RoboDK station: 6640_station.rdk

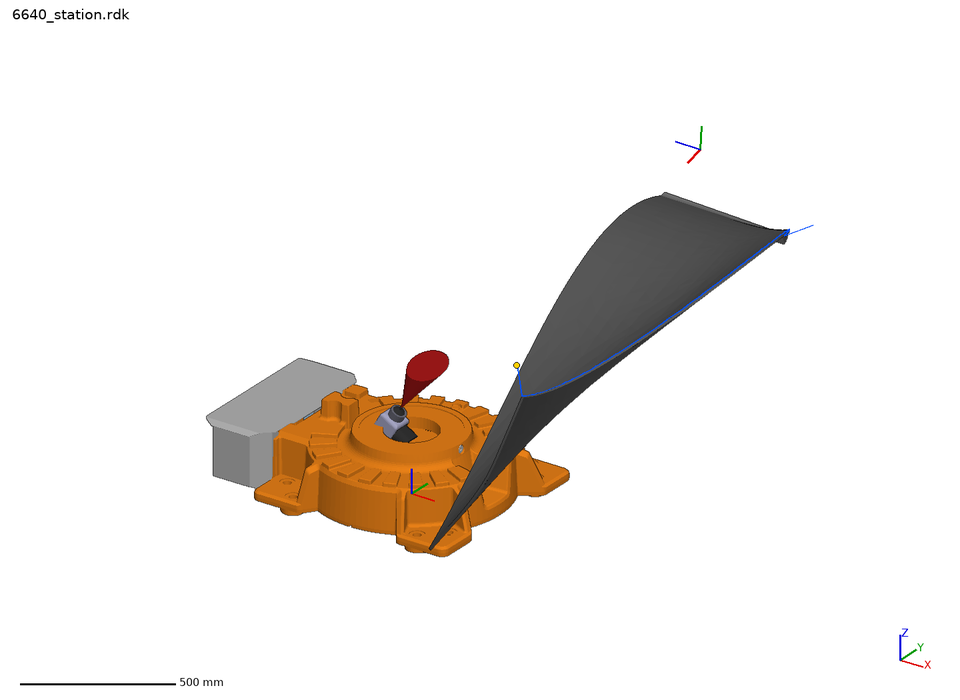
[picture v0: the station drawn from its stored meshes, robots at their saved joint values, targets as dots, program paths as lines]
Station 6640_station (saved by RoboDK 5.3.2). Poses are relative to the parent item; angles as X-Y-Z fixed-axis rotations.
  - frame Frame 2 at (435.15, 997.23, 955.19) mm, rotated rx 84.12 ry 5.86 rz -82.67 deg
    - object Curve_sparse at (0, 0, 0) mm
    - object generic_fan_blade at (0, 0, 0) mm, size 1633.1 x 757.5 x 617.2 mm, 1 curves, geometry from generic_fan_blade.igs
  - machining project Path1 settings: rotZ(0) | rotX(0)*rotY(0) | rotz(0)
  - program Path1 (113 instructions, listed below)
  - frame ABB IRB 6640-180/2.55 Base at (0, 0, 0) mm
    - robot ABB IRB 6640-180/2.55: 6 axes, payload 180 kg, reach 2550 mm, repeatability 0.07 mm, weight 1310 kg
        joint limits [-170, -65, -180, -300, -120, -360] to [170, 85, 70, 300, 120, 360]; home [0, 0, 0, 0, 0, 0]; saved at [53.767, 31.077, 10.307, -34.616, 114.864, 62.566]
      - tool Paint gun, TCP at (75, 0, 493.3) mm, rotated rx 0 ry 30 rz 0 deg, size 203.2 x 279.7 x 471.5 mm
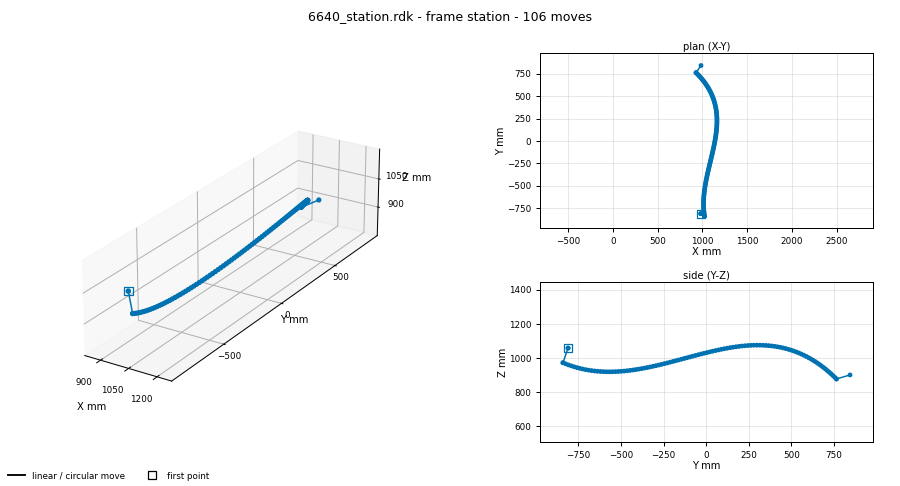
[picture p0: tool path of 6640_station.rdk in frame station, 106 of 106 moves have a stored position in this frame; points joined in program order, loops and branches not executed]

--- program Path1 (robot ABB IRB 6640-180/2.55) ---
  Smooth(1)
  Set speed (500.0 mm/s)
  Set Ref.: Frame 2
  Set Tool: Paint gun
  Show Paint gun
  MoveJ 1 to (1843, 323.42, -278.71) mm, rotated rx -160.29 ry -61.06 rz -82.99 deg; joints [-55.097, -38.535, 54.626, 57.641, 41.418, -99.137]
  MoveL 2 to (1843, 323.42, -278.71) mm, rotated rx -160.29 ry -61.06 rz -82.99 deg; joints [-55.097, -38.535, 54.626, 57.641, 41.418, -99.137]
  MoveL 3 to (1886.54, 245.77, -324.26) mm, rotated rx -160.29 ry -61.06 rz -82.99 deg; joints [-53.957, -33.784, 56.818, 64.848, 37.125, -107.941]
  MoveL 4 to (1886.54, 245.77, -324.26) mm, rotated rx -160.29 ry -61.06 rz -82.99 deg; joints [-53.957, -33.784, 56.818, 64.848, 37.125, -107.941]
  Set speed (50.0 mm/s)
  MoveL 5 to (1871.02, 237.56, -324.78) mm, rotated rx -160.62 ry -60.74 rz -83.73 deg; joints [-53.875, -34.314, 57.338, 64.8, 37.71, -106.973]
  MoveL 6 to (1855.29, 229.78, -325.6) mm, rotated rx -160.63 ry -60.92 rz -84.77 deg; joints [-53.458, -34.858, 57.629, 63.666, 37.945, -104.885]
  MoveL 7 to (1839.38, 222.45, -326.7) mm, rotated rx -160.51 ry -61.31 rz -85.95 deg; joints [-52.891, -35.379, 57.794, 62.071, 38.083, -102.301]
  MoveL 8 to (1823.28, 215.57, -328.1) mm, rotated rx -160.35 ry -61.75 rz -87.2 deg; joints [-52.27, -35.863, 57.894, 60.357, 38.247, -99.564]
  MoveL 9 to (1807.02, 209.15, -329.78) mm, rotated rx -160.22 ry -62.19 rz -88.46 deg; joints [-51.64, -36.309, 57.963, 58.692, 38.477, -96.847]
  MoveL 10 to (1790.62, 203.19, -331.75) mm, rotated rx -160.11 ry -62.58 rz -89.71 deg; joints [-51.014, -36.722, 58.014, 57.137, 38.778, -94.214]
  MoveL 11 to (1774.08, 197.71, -334) mm, rotated rx -160.03 ry -62.95 rz -90.94 deg; joints [-50.391, -37.105, 58.048, 55.697, 39.138, -91.674]
  MoveL 12 to (1757.44, 192.71, -336.52) mm, rotated rx -159.97 ry -63.29 rz -92.16 deg; joints [-49.767, -37.458, 58.065, 54.358, 39.543, -89.215]
  MoveL 13 to (1740.71, 188.17, -339.31) mm, rotated rx -159.93 ry -63.62 rz -93.37 deg; joints [-49.135, -37.783, 58.062, 53.107, 39.982, -86.827]
  MoveL 14 to (1723.9, 184.11, -342.35) mm, rotated rx -159.91 ry -63.94 rz -94.57 deg; joints [-48.493, -38.081, 58.041, 51.935, 40.446, -84.505]
  MoveL 15 to (1707.03, 180.51, -345.64) mm, rotated rx -159.9 ry -64.25 rz -95.74 deg; joints [-47.841, -38.354, 58.002, 50.844, 40.929, -82.253]
  MoveL 16 to (1690.11, 177.36, -349.16) mm, rotated rx -159.91 ry -64.54 rz -96.89 deg; joints [-47.181, -38.607, 57.951, 49.84, 41.423, -80.08]
  MoveL 17 to (1673.17, 174.65, -352.91) mm, rotated rx -159.93 ry -64.82 rz -98 deg; joints [-46.514, -38.843, 57.892, 48.927, 41.92, -77.993]
  MoveL 18 to (1656.22, 172.37, -356.87) mm, rotated rx -159.97 ry -65.08 rz -99.08 deg; joints [-45.841, -39.067, 57.83, 48.104, 42.414, -75.993]
  MoveL 19 to (1639.26, 170.51, -361.03) mm, rotated rx -160.03 ry -65.31 rz -100.1 deg; joints [-45.161, -39.285, 57.767, 47.369, 42.896, -74.079]
  MoveL 20 to (1622.3, 169.06, -365.37) mm, rotated rx -160.12 ry -65.52 rz -101.08 deg; joints [-44.472, -39.497, 57.703, 46.71, 43.36, -72.243]
  MoveL 21 to (1605.37, 167.99, -369.89) mm, rotated rx -160.21 ry -65.72 rz -102.02 deg; joints [-43.772, -39.707, 57.639, 46.115, 43.802, -70.472]
  MoveL 22 to (1588.46, 167.28, -374.56) mm, rotated rx -160.31 ry -65.9 rz -102.91 deg; joints [-43.056, -39.912, 57.571, 45.567, 44.218, -68.753]
  MoveL 23 to (1571.57, 166.93, -379.39) mm, rotated rx -160.42 ry -66.08 rz -103.76 deg; joints [-42.322, -40.111, 57.497, 45.052, 44.607, -67.07]
  MoveL 24 to (1554.73, 166.92, -384.35) mm, rotated rx -160.52 ry -66.26 rz -104.59 deg; joints [-41.567, -40.302, 57.413, 44.554, 44.969, -65.412]
  MoveL 25 to (1537.92, 167.22, -389.43) mm, rotated rx -160.62 ry -66.44 rz -105.39 deg; joints [-40.788, -40.481, 57.315, 44.061, 45.306, -63.767]
  MoveL 26 to (1521.16, 167.82, -394.63) mm, rotated rx -160.7 ry -66.64 rz -106.16 deg; joints [-39.985, -40.646, 57.2, 43.565, 45.618, -62.128]
  MoveL 27 to (1504.44, 168.7, -399.93) mm, rotated rx -160.77 ry -66.85 rz -106.93 deg; joints [-39.156, -40.793, 57.067, 43.059, 45.908, -60.489]
  MoveL 28 to (1487.77, 169.85, -405.32) mm, rotated rx -160.81 ry -67.07 rz -107.68 deg; joints [-38.303, -40.92, 56.914, 42.54, 46.178, -58.848]
  MoveL 29 to (1471.14, 171.25, -410.79) mm, rotated rx -160.84 ry -67.31 rz -108.42 deg; joints [-37.425, -41.027, 56.741, 42.003, 46.429, -57.204]
  MoveL 30 to (1454.56, 172.87, -416.33) mm, rotated rx -160.85 ry -67.57 rz -109.15 deg; joints [-36.523, -41.112, 56.547, 41.45, 46.662, -55.556]
  MoveL 31 to (1438.02, 174.71, -421.93) mm, rotated rx -160.84 ry -67.85 rz -109.87 deg; joints [-35.599, -41.175, 56.332, 40.879, 46.88, -53.905]
  MoveL 32 to (1421.52, 176.76, -427.59) mm, rotated rx -160.8 ry -68.15 rz -110.58 deg; joints [-34.653, -41.215, 56.098, 40.289, 47.083, -52.251]
  MoveL 33 to (1405.07, 178.98, -433.29) mm, rotated rx -160.74 ry -68.46 rz -111.29 deg; joints [-33.687, -41.233, 55.843, 39.681, 47.273, -50.595]
  MoveL 34 to (1388.64, 181.38, -439.03) mm, rotated rx -160.65 ry -68.79 rz -111.99 deg; joints [-32.7, -41.226, 55.57, 39.054, 47.452, -48.938]
  MoveL 35 to (1372.25, 183.93, -444.79) mm, rotated rx -160.53 ry -69.13 rz -112.69 deg; joints [-31.695, -41.197, 55.277, 38.407, 47.62, -47.278]
  MoveL 36 to (1355.89, 186.62, -450.58) mm, rotated rx -160.38 ry -69.49 rz -113.38 deg; joints [-30.672, -41.144, 54.965, 37.74, 47.779, -45.618]
  MoveL 37 to (1339.56, 189.43, -456.38) mm, rotated rx -160.21 ry -69.87 rz -114.08 deg; joints [-29.632, -41.067, 54.635, 37.053, 47.93, -43.956]
  MoveL 38 to (1323.25, 192.36, -462.18) mm, rotated rx -160 ry -70.26 rz -114.78 deg; joints [-28.575, -40.967, 54.287, 36.345, 48.075, -42.293]
  MoveL 39 to (1306.95, 195.39, -467.98) mm, rotated rx -159.75 ry -70.66 rz -115.49 deg; joints [-27.502, -40.844, 53.922, 35.616, 48.215, -40.629]
  MoveL 40 to (1290.67, 198.51, -473.78) mm, rotated rx -159.46 ry -71.08 rz -116.19 deg; joints [-26.414, -40.7, 53.54, 34.866, 48.349, -38.964]
  MoveL 41 to (1274.4, 201.7, -479.55) mm, rotated rx -159.13 ry -71.51 rz -116.91 deg; joints [-25.311, -40.534, 53.143, 34.094, 48.48, -37.298]
  MoveL 42 to (1258.13, 204.96, -485.31) mm, rotated rx -158.76 ry -71.95 rz -117.64 deg; joints [-24.193, -40.348, 52.731, 33.299, 48.607, -35.631]
  MoveL 43 to (1241.86, 208.26, -491.03) mm, rotated rx -158.34 ry -72.4 rz -118.38 deg; joints [-23.06, -40.142, 52.305, 32.48, 48.731, -33.961]
  MoveL 44 to (1225.59, 211.59, -496.72) mm, rotated rx -157.87 ry -72.86 rz -119.13 deg; joints [-21.913, -39.918, 51.865, 31.635, 48.854, -32.288]
  MoveL 45 to (1209.31, 214.96, -502.37) mm, rotated rx -157.34 ry -73.33 rz -119.91 deg; joints [-20.751, -39.674, 51.411, 30.762, 48.976, -30.609]
  MoveL 46 to (1193.01, 218.33, -507.96) mm, rotated rx -156.74 ry -73.81 rz -120.72 deg; joints [-19.573, -39.41, 50.943, 29.859, 49.101, -28.923]
  MoveL 47 to (1176.7, 221.7, -513.5) mm, rotated rx -156.06 ry -74.3 rz -121.57 deg; joints [-18.38, -39.125, 50.46, 28.924, 49.23, -27.228]
  MoveL 48 to (1160.36, 225.06, -518.97) mm, rotated rx -155.3 ry -74.8 rz -122.47 deg; joints [-17.171, -38.817, 49.96, 27.954, 49.368, -25.521]
  MoveL 49 to (1143.99, 228.39, -524.37) mm, rotated rx -154.43 ry -75.31 rz -123.43 deg; joints [-15.945, -38.485, 49.444, 26.947, 49.517, -23.803]
  MoveL 50 to (1127.58, 231.68, -529.68) mm, rotated rx -153.43 ry -75.84 rz -124.48 deg; joints [-14.703, -38.128, 48.909, 25.901, 49.682, -22.07]
  MoveL 51 to (1111.14, 234.91, -534.91) mm, rotated rx -152.29 ry -76.39 rz -125.63 deg; joints [-13.443, -37.744, 48.356, 24.815, 49.865, -20.322]
  MoveL 52 to (1094.65, 238.08, -540.05) mm, rotated rx -150.98 ry -76.94 rz -126.9 deg; joints [-12.166, -37.332, 47.783, 23.688, 50.069, -18.558]
  MoveL 53 to (1078.12, 241.17, -545.07) mm, rotated rx -149.48 ry -77.51 rz -128.33 deg; joints [-10.869, -36.894, 47.192, 22.517, 50.296, -16.776]
  MoveL 54 to (1061.53, 244.16, -549.99) mm, rotated rx -147.74 ry -78.08 rz -129.93 deg; joints [-9.554, -36.43, 46.584, 21.302, 50.548, -14.977]
  MoveL 55 to (1044.89, 247.05, -554.77) mm, rotated rx -145.74 ry -78.65 rz -131.75 deg; joints [-8.217, -35.94, 45.959, 20.042, 50.825, -13.157]
  MoveL 56 to (1028.18, 249.8, -559.43) mm, rotated rx -143.44 ry -79.22 rz -133.81 deg; joints [-6.858, -35.426, 45.32, 18.734, 51.128, -11.317]
  MoveL 57 to (1011.42, 252.41, -563.94) mm, rotated rx -140.79 ry -79.78 rz -136.17 deg; joints [-5.475, -34.889, 44.668, 17.377, 51.457, -9.454]
  MoveL 58 to (994.59, 254.86, -568.29) mm, rotated rx -137.74 ry -80.32 rz -138.86 deg; joints [-4.066, -34.331, 44.004, 15.968, 51.814, -7.566]
  MoveL 59 to (977.7, 257.14, -572.47) mm, rotated rx -134.25 ry -80.84 rz -141.93 deg; joints [-2.631, -33.752, 43.33, 14.505, 52.2, -5.65]
  MoveL 60 to (960.73, 259.22, -576.48) mm, rotated rx -130.25 ry -81.31 rz -145.43 deg; joints [-1.166, -33.15, 42.647, 12.986, 52.617, -3.707]
  MoveL 61 to (943.7, 261.09, -580.29) mm, rotated rx -125.71 ry -81.74 rz -149.4 deg; joints [0.328, -32.525, 41.955, 11.411, 53.071, -1.733]
  MoveL 62 to (926.6, 262.73, -583.9) mm, rotated rx -120.59 ry -82.12 rz -153.88 deg; joints [1.854, -31.875, 41.255, 9.778, 53.564, 0.271]
  MoveL 63 to (909.44, 264.11, -587.29) mm, rotated rx -114.89 ry -82.42 rz -158.86 deg; joints [3.412, -31.196, 40.547, 8.088, 54.104, 2.305]
  MoveL 64 to (892.21, 265.22, -590.45) mm, rotated rx -108.65 ry -82.63 rz -164.3 deg; joints [5.002, -30.488, 39.831, 6.342, 54.694, 4.368]
  MoveL 65 to (874.92, 266.04, -593.36) mm, rotated rx -102 ry -82.75 rz -170.06 deg; joints [6.624, -29.747, 39.109, 4.543, 55.339, 6.458]
  MoveL 66 to (857.57, 266.55, -596) mm, rotated rx -95.12 ry -82.76 rz -175.97 deg; joints [8.279, -28.973, 38.381, 2.694, 56.043, 8.572]
  MoveL 67 to (840.18, 266.73, -598.37) mm, rotated rx -88.24 ry -82.65 rz 178.22 deg; joints [9.965, -28.163, 37.652, 0.799, 56.808, 10.708]
  MoveL 68 to (822.75, 266.54, -600.45) mm, rotated rx -81.6 ry -82.44 rz 172.75 deg; joints [11.681, -27.319, 36.924, -1.137, 57.637, 12.86]
  MoveL 69 to (805.3, 265.99, -602.22) mm, rotated rx -75.41 ry -82.12 rz 167.81 deg; joints [13.425, -26.439, 36.201, -3.106, 58.53, 15.025]
  MoveL 70 to (787.84, 265.04, -603.67) mm, rotated rx -69.79 ry -81.71 rz 163.55 deg; joints [15.194, -25.523, 35.487, -5.102, 59.486, 17.197]
  MoveL 71 to (770.37, 263.68, -604.78) mm, rotated rx -64.79 ry -81.22 rz 160 deg; joints [16.983, -24.572, 34.786, -7.116, 60.505, 19.368]
  MoveL 72 to (752.93, 261.89, -605.55) mm, rotated rx -60.41 ry -80.68 rz 157.15 deg; joints [18.788, -23.585, 34.102, -9.137, 61.587, 21.53]
  MoveL 73 to (735.53, 259.66, -605.96) mm, rotated rx -56.59 ry -80.09 rz 154.96 deg; joints [20.601, -22.561, 33.436, -11.153, 62.731, 23.675]
  MoveL 74 to (718.19, 256.98, -606) mm, rotated rx -53.27 ry -79.47 rz 153.35 deg; joints [22.417, -21.497, 32.792, -13.152, 63.935, 25.792]
  MoveL 75 to (700.94, 253.83, -605.66) mm, rotated rx -50.36 ry -78.83 rz 152.23 deg; joints [24.226, -20.393, 32.169, -15.119, 65.198, 27.871]
  MoveL 76 to (683.78, 250.21, -604.94) mm, rotated rx -47.79 ry -78.17 rz 151.53 deg; joints [26.021, -19.246, 31.568, -17.041, 66.517, 29.903]
  MoveL 77 to (666.76, 246.11, -603.84) mm, rotated rx -45.51 ry -77.49 rz 151.18 deg; joints [27.792, -18.054, 30.988, -18.904, 67.89, 31.878]
  MoveL 78 to (649.88, 241.54, -602.35) mm, rotated rx -43.44 ry -76.8 rz 151.11 deg; joints [29.532, -16.817, 30.429, -20.696, 69.313, 33.788]
  MoveL 79 to (633.17, 236.5, -600.48) mm, rotated rx -41.55 ry -76.09 rz 151.26 deg; joints [31.231, -15.531, 29.887, -22.404, 70.783, 35.626]
  MoveL 80 to (616.66, 230.99, -598.23) mm, rotated rx -39.79 ry -75.37 rz 151.59 deg; joints [32.883, -14.196, 29.36, -24.02, 72.297, 37.386]
  MoveL 81 to (600.36, 225.03, -595.61) mm, rotated rx -38.12 ry -74.63 rz 152.04 deg; joints [34.48, -12.809, 28.842, -25.533, 73.852, 39.065]
  MoveL 82 to (584.29, 218.62, -592.63) mm, rotated rx -36.52 ry -73.86 rz 152.6 deg; joints [36.016, -11.366, 28.328, -26.936, 75.447, 40.66]
  MoveL 83 to (568.46, 211.78, -589.29) mm, rotated rx -34.96 ry -73.05 rz 153.23 deg; joints [37.486, -9.867, 27.815, -28.224, 77.081, 42.172]
  MoveL 84 to (552.91, 204.52, -585.61) mm, rotated rx -33.43 ry -72.21 rz 153.93 deg; joints [38.885, -8.31, 27.296, -29.395, 78.751, 43.601]
  MoveL 85 to (537.62, 196.87, -581.6) mm, rotated rx -31.92 ry -71.31 rz 154.67 deg; joints [40.212, -6.698, 26.771, -30.446, 80.453, 44.952]
  MoveL 86 to (522.62, 188.84, -577.28) mm, rotated rx -30.45 ry -70.38 rz 155.47 deg; joints [41.464, -5.035, 26.24, -31.381, 82.18, 46.231]
  MoveL 87 to (507.91, 180.46, -572.66) mm, rotated rx -29.03 ry -69.4 rz 156.33 deg; joints [42.642, -3.329, 25.704, -32.204, 83.922, 47.445]
  MoveL 88 to (493.49, 171.73, -567.76) mm, rotated rx -27.66 ry -68.39 rz 157.26 deg; joints [43.748, -1.59, 25.168, -32.921, 85.669, 48.603]
  MoveL 89 to (479.36, 162.69, -562.59) mm, rotated rx -26.35 ry -67.35 rz 158.25 deg; joints [44.785, 0.174, 24.636, -33.539, 87.412, 49.712]
  MoveL 90 to (465.53, 153.35, -557.16) mm, rotated rx -25.11 ry -66.3 rz 159.3 deg; joints [45.754, 1.957, 24.108, -34.063, 89.146, 50.779]
  MoveL 91 to (451.98, 143.72, -551.51) mm, rotated rx -23.91 ry -65.21 rz 160.41 deg; joints [46.658, 3.76, 23.581, -34.499, 90.874, 51.811]
  MoveL 92 to (438.73, 133.83, -545.62) mm, rotated rx -22.76 ry -64.09 rz 161.56 deg; joints [47.498, 5.584, 23.054, -34.847, 92.6, 52.813]
  MoveL 93 to (425.75, 123.7, -539.53) mm, rotated rx -21.64 ry -62.94 rz 162.77 deg; joints [48.275, 7.433, 22.521, -35.112, 94.329, 53.793]
  MoveL 94 to (413.06, 113.33, -533.24) mm, rotated rx -20.56 ry -61.74 rz 164.03 deg; joints [48.991, 9.304, 21.984, -35.296, 96.062, 54.756]
  MoveL 95 to (400.64, 102.75, -526.77) mm, rotated rx -19.52 ry -60.52 rz 165.34 deg; joints [49.648, 11.188, 21.447, -35.405, 97.793, 55.711]
  MoveL 96 to (388.49, 91.97, -520.13) mm, rotated rx -18.52 ry -59.28 rz 166.7 deg; joints [50.253, 13.076, 20.916, -35.446, 99.511, 56.663]
  MoveL 97 to (376.59, 81, -513.32) mm, rotated rx -17.57 ry -58.02 rz 168.12 deg; joints [50.808, 14.961, 20.395, -35.424, 101.212, 57.617]
  MoveL 98 to (364.95, 69.86, -506.37) mm, rotated rx -16.66 ry -56.76 rz 169.58 deg; joints [51.317, 16.845, 19.884, -35.345, 102.902, 58.581]
  MoveL 99 to (353.55, 58.56, -499.27) mm, rotated rx -15.79 ry -55.49 rz 171.1 deg; joints [51.783, 18.726, 19.383, -35.212, 104.58, 59.559]
  MoveL 100 to (342.39, 47.11, -492.05) mm, rotated rx -14.97 ry -54.24 rz 172.66 deg; joints [52.213, 20.583, 18.906, -35.031, 106.222, 60.551]
  MoveL 101 to (331.46, 35.51, -484.7) mm, rotated rx -14.21 ry -53.06 rz 174.23 deg; joints [52.619, 22.372, 18.471, -34.812, 107.78, 61.549]
  MoveL 102 to (320.75, 23.78, -477.23) mm, rotated rx -13.5 ry -51.95 rz 175.8 deg; joints [53.005, 24.107, 18.073, -34.559, 109.266, 62.554]
  MoveL 103 to (310.26, 11.94, -469.66) mm, rotated rx -12.77 ry -50.75 rz 177.49 deg; joints [53.342, 25.914, 17.654, -34.254, 110.839, 63.61]
  MoveL 104 to (300, 0, -462) mm, rotated rx -12.21 ry -49.81 rz 178.85 deg; joints [53.682, 27.418, 17.334, -33.873, 112.045, 64.577]
  Set speed (500.0 mm/s)
  MoveL 105 to (300, 0, -462) mm, rotated rx -12.21 ry -49.81 rz 178.85 deg; joints [53.682, 27.418, 17.334, -33.873, 112.045, 64.577]
  MoveL 106 to (225.78, 22.65, -525.08) mm, rotated rx -12.21 ry -49.81 rz 178.85 deg; joints [53.767, 31.077, 10.307, -34.616, 114.864, 62.566]
